// TIA Portal V19 export
DATA_BLOCK "BACKWACH DB"   // DB80
{ S7_Optimized_Access := 'FALSE' }
   VAR
      "BACKWASH_TIMER SET" : Int;
      "BACKWASH_TIMER PV" : Int;
      OUTPUT : Struct
         "ABFV-102" : Bool;
         "ABFV-103" : Bool;
         "BACK WASH RECOVERY P-801 A" : Bool;
         "BACK WASH RECOVERY P-801 B" : Bool;
      END_STRUCT;
   END_VAR
BEGIN
END_DATA_BLOCK
